Staubli VAL3: Offset.pgx

program Offset(trsf& x_trOffset)
  local bool l_bRes
  local num l_i
  local num l_nKey
  local num l_nSelect
  local string l_sItem
  local string l_sValue
begin
  cls()
  resize(sParameter,1,3)
  sParameter[0]="X"
  sParameter[1]="Y"
  sParameter[2]="Z"
  resize(sListItemValue,1,size(sParameter))
  sListItemValue[0]=toString(".2",x_trOffset.x)
  sListItemValue[1]=toString(".2",x_trOffset.y)
  sListItemValue[2]=toString(".2",x_trOffset.z)

  //增加变量
  for l_i=0 to size(sParameter)-1
    call user:strlength(sParameter[l_i],user:nBottomX/2)
    l_sValue=sListItemValue[l_i]
    call user:strlength(l_sValue,user:nBottomX/2+1)
    sParameter[l_i]=sParameter[l_i]+":"+l_sValue
  endFor

  bUserRefresh=true
  bListRefresh=true
  //
  do
    if bUserRefresh
      cls()
      call user:clear(0,13)
      call user:typeMenu(8,"确定")
    endIf
    call user:setList("偏移",sParameter,bUserRefresh,bListRefresh,l_nSelect,l_sItem,l_nKey)
    bUserRefresh=false
    bListRefresh=false
    call EnterPageKey(l_nKey,l_nSelect,sParameter[l_nSelect],x_trOffset)
    delay(0)
  until l_nKey==255 or l_nKey==278
  fFrmTemp.trsf=frmaster.trsf*trOffset
  bUserRefresh=true
  bListRefresh=true
end
